FUNCTION_BLOCK FbDelayN (* Блок задержки сигнала на 100 тактов. *)
  (* Standard: 61499-1; Description: Блок задержки сигнала на 100 тактов. Simple FB with one algorithm *)
  (* Version 2.3, 2026-03-22, VA, LIB_PLC *)
  (* Documentation:
  // Блок задержки сигнала на 100 тактов. //      DbDelayN //    +----------+ //    | FbDelayN | // ->-|In     Out|->- //    +----------+
  *)
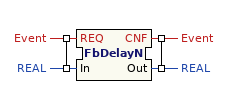
  EVENT_INPUT
    REQ WITH In; (* Normal Execution Request *)
  END_EVENT
  EVENT_OUTPUT
    CNF WITH Out; (* Execution Confirmation *)
  END_EVENT
  VAR_INPUT
    In : REAL := 0.0; (* Вход. *)
  END_VAR
  VAR_OUTPUT
    Out : REAL := 0.0; (* Выход. *)
  END_VAR
  VAR CONSTANT
    NUMBER : INT := 98; (* Размер массива Тактов 100 - 2 = 98. *)
  END_VAR
  VAR
    Buffer1 : ARRAY [0..NUMBER] OF REAL; (* Буфер задержки сигнала. *)
  END_VAR
  EC_STATES
    REQ : REQ -> CNF;
  END_STATES
  ALGORITHM REQ IN ST:
VAR_TEMP
	Counter1 : INT := 0; // Счетчик.
END_VAR

// W(Z)=Z^(-N), N=NUMBER+2
Out := Buffer1[NUMBER];
FOR Counter1 := NUMBER TO 1 BY -1 DO
	Buffer1[Counter1] := Buffer1[Counter1 - 1];
END_FOR;
Buffer1[0] := In;

// @COPYLEFT ALL WRONGS RESERVED :)
// Author: VA
// Contacts: DIY.PLC.314@gmail.com
// Date start LIB_PLC: 2014
// License: GNU GPL-2.0-or-later
// https://www.gnu.org/licenses/old-licenses/gpl-2.0.html
// https://www.youtube.com/watch?v=n1F_MfLRlX0
// https://www.youtube.com/@DIY_PLC
// https://github.com/DIYPLC/LIB_PLC
// https://oshwlab.com/diy.plc.314/PLC_HW1_SW1
// https://3dtoday.ru/3d-models/mechanical-parts/body/korpus-na-din-reiku
// https://t.me/DIY_PLC
  END_ALGORITHM
END_FUNCTION_BLOCK
